// TIA Portal V15.1 export
// export: Created 2026-01-15T16:29:45.9870454Z, ExportSetting WithDefaults, WithReadOnly, DisplayName Totally Integrated Automation Portal, DisplayVersion V15.1 Update 8, DisplayName TIA Portal Openness, DisplayVersion V15.1 Update 8, DisplayName STEP 7 Professional, DisplayVersion V15.1 Update 8, DisplayName WinCC Advanced, DisplayVersion V15.1 Update 8
DATA_BLOCK "C#3_WD_SILO"   // DB3
{ S7_Optimized_Access := 'FALSE' }
VERSION : 0.1
// stored: AutoNumber true, CodeModifiedDate 2024-09-25T15:44:48.8692886Z, CompileDate 2026-01-15T16:25:51.9840274Z, CreationDate 2026-01-15T16:23:32.6582836Z, DBAccessibleFromOPCUA true, InterfaceModifiedDate 2024-09-25T15:44:48.8692886Z, IsConsistent true, IsKnowHowProtected false, IsOnlyStoredInLoadMemory false, IsPLCDB false, IsWriteProtectedInAS false, ModifiedDate 2024-09-25T15:47:56.1309792Z, ParameterModified 2024-09-25T15:44:48.8692886Z, StructureModified 2024-09-25T15:44:48.8692886Z
   VAR RETAIN
      AG1_SS_TREN : Real;   // Ag1 sai số trên
      AG1_SS_DUOI : Real;   // Ag1 sai số dưới
      AG1_KL_RTD : Real;   // Ag1 khối lượng rơi tự do
      AG1_TG_ON_CAN : Real;   // Ag1 thời gian mở cân
      AG1_TG_OFF_CAN : Real;   // Ag1 thời gian đóng cân
      AG1_TG_ODC : Real;   // Ag1 thời gian tính lượng rơi thêm
      AG2_SS_TREN : Real;   // Ag2 sai số trên
      AG2_SS_DUOI : Real;   // Ag2 sai số dưới
      AG2_KL_RTD : Real;   // Ag2 khối lượng rơi tự do
      AG2_TG_ON_CAN : Real;   // Ag2 thời gian mở cân
      AG2_TG_OFF_CAN : Real;   // Ag2 thời gian đóng cân
      AG2_TG_ODC : Real;   // Ag2 thời gian tính lượng rơi thêm
      AG3_SS_TREN : Real;   // Ag3 sai số trên
      AG3_SS_DUOI : Real;   // Ag3 sai số dưới
      AG3_KL_RTD : Real;   // Ag3 khối lượng rơi tự do
      AG3_TG_ON_CAN : Real;   // Ag3 thời gian mở cân
      AG3_TG_OFF_CAN : Real;   // Ag3 thời gian đóng cân
      AG3_TG_ODC : Real;   // Ag3 thời gian tính lượng rơi thêm
      AG4_SS_TREN : Real;   // Ag4 sai số trên
      AG4_SS_DUOI : Real;   // Ag4 sai số dưới
      AG4_KL_RTD : Real;   // Ag4 khối lượng rơi tự do
      AG4_TG_ON_CAN : Real;   // Ag4 thời gian mở cân
      AG4_TG_OFF_CAN : Real;   // Ag4 thời gian đóng cân
      AG4_TG_ODC : Real;   // Ag4 thời gian tính lượng rơi thêm
      AG5_SS_TREN : Real;   // Ag5 sai số trên
      AG5_SS_DUOI : Real;   // Ag5 sai số dưới
      AG5_KL_RTD : Real;   // Ag5 khối lượng rơi tự do
      AG5_TG_ON_CAN : Real;   // Ag5 thời gian mở cân
      AG5_TG_OFF_CAN : Real;   // Ag5 thời gian đóng cân
      AG5_TG_ODC : Real;   // Ag5 thời gian tính lượng rơi thêm
      FD1_SS_TREN : Real;   // FD1 sai số trên
      FD1_SS_DUOI : Real;   // FD1 sai số dưới
      FD1_KL_RTD : Real;   // FD1 khối lượng rơi tự do
      FD1_TG_ON_CAN : Real;   // FD1 thời gian mở cân
      FD1_TG_OFF_CAN : Real;   // FD1 thời gian đóng cân
      FD1_TG_ODC : Real;   // FD1 thời gian tính lượng rơi thêm
      AP1_SS_TREN : Real;   // AP1 sai số trên
      AP1_SS_DUOI : Real;   // AP1 sai số dưới
      AP1_KL_RTD : Real;   // AP1 khối lượng rơi tự do
      AP1_TG_ON_CAN : Real;   // AP1 thời gian mở cân
      AP1_TG_OFF_CAN : Real;   // AP1 thời gian đóng cân
      AP1_TG_ODC : Real;   // AP1 thời gian tính lượng rơi thêm
      SB1_SS_TREN : Real;   // SBS1 sai số trên
      SB1_SS_DUOI : Real;   // SBS1 sai số dưới
      SB1_KL_RTD : Real;   // SBS1 khối lượng rơi tự do
      SB1_TG_ON_CAN : Real;   // SBS1 thời gian mở cân
      SB1_TG_OFF_CAN : Real;   // SBS1 thời gian đóng cân
      SB1_TG_ODC : Real;   // SBS1 thời gian tính lượng rơi thêm
   END_VAR
BEGIN
END_DATA_BLOCK
